Fanuc KAREL source: kf00081.KL

-- PROVISIONAL review KL for V770-1; original PC SHA256 b2409d5a0a957c4a85f80cb925038a58fc2b2f9a8b872979cc4209381c6d70fc
-- Incomplete behavior may be omitted. Consult companion uncertainty JSON. Do not deploy.
PROGRAM KF00081
%NOLOCKGROUP
BEGIN
  -- UNRESOLVED_PC offsets 5-15; opcodes 27,22,31
  -- UNRESOLVED_PC offsets 20-54; opcodes 27,27,2E,22,22,22,22,31
  -- UNRESOLVED_PC offsets 59-63; opcodes 7F
END KF00081
